(* CoDeSys 2.3 export: INIT.EXP *)

(* POU INIT, ST *)
PROGRAM INIT
VAR
END_VAR

END_PROGRAM
